Yaskawa INFORM job: TATTRACE.JBI

/JOB
//NAME TATTRACE
//POS
///NPOS 22,0,0,0,0,0
///TOOL 0
///POSTYPE PULSE
///PULSE
C00000=-2822,58859,-1118,-1041,-34109,-89
C00001=-2466,58809,-1226,-1089,-34047,-231
C00002=-2724,58654,-1466,-1058,-33950,-125
C00003=-2857,58313,-1983,-1045,-33743,-68
C00004=-2875,57908,-2594,-1049,-33498,-56
C00005=-2788,57537,-3152,-1066,-33274,-86
C00006=-2630,57202,-3656,-1092,-33070,-146
C00007=-2429,56890,-4127,-1124,-32879,-222
C00008=-2203,56625,-4527,-1158,-32716,-309
C00009=-1962,56480,-4747,-1193,-32624,-403
C00010=-1717,56689,-4430,-1223,-32750,-504
C00011=-1489,56956,-4022,-1249,-32913,-598
C00012=-1286,57250,-3573,-1271,-33094,-684
C00013=-1137,57578,-3072,-1285,-33296,-748
C00014=-1063,57950,-2503,-1288,-33527,-783
C00015=-1110,58338,-1911,-1275,-33768,-770
C00016=-1288,58654,-1434,-1246,-33962,-703
C00017=-1567,58754,-1289,-1207,-34021,-593
C00018=-1829,58620,-1499,-1175,-33936,-485
C00019=-1996,58422,-1802,-1157,-33814,-415
C00020=-2184,58721,-1353,-1127,-33995,-343
C00021=-2466,58809,-1226,-1089,-34047,-231
//INST
///DATE 2026/04/15 15:34
///ATTR SC,RW
///GROUP1 RB1
NOP
MOVJ C00000 VJ=0.78
MOVJ C00001 VJ=0.78
MOVJ C00002 VJ=0.78
MOVJ C00003 VJ=0.78
MOVJ C00004 VJ=0.78
MOVJ C00005 VJ=0.78
MOVJ C00006 VJ=0.78
MOVJ C00007 VJ=0.78
MOVJ C00008 VJ=0.78
MOVJ C00009 VJ=0.78
MOVJ C00010 VJ=0.78
MOVJ C00011 VJ=0.78
MOVJ C00012 VJ=0.78
MOVJ C00013 VJ=0.78
MOVJ C00014 VJ=0.78
MOVJ C00015 VJ=0.78
MOVJ C00016 VJ=0.78
MOVJ C00017 VJ=0.78
MOVJ C00018 VJ=0.78
MOVJ C00019 VJ=0.78
MOVJ C00020 VJ=0.78
MOVJ C00021 VJ=0.78
END
